PROGRAM MAIN
VAR
	test_bool:BOOL;
	test_int:INT;
	test_real:REAL;
	test_string:STRING;
	test_arr_int:ARRAY[1..10] OF INT;
	test_word:WORD;
	test_arr_bool:ARRAY[1..3] OF BOOL;
	test_structure:user_defined_structure;
	test_arr_string:ARRAY[1..3] OF STRING;
	
	fb_Time : FB_LocalSystemTime;

	byte1 : BYTE;
	string1 :STRING;

	
END_VAR

fb_Time(bEnable := TRUE); 

M_mappingIO();
M_measuringLC();
M_rfid();
runEveryCycle();
M_ReM();

METHOD M_mappingIO 
VAR_INPUT
END_VAR
GVL.fb_remIOmapping[0](iReM:= 0);
GVL.fb_remIOmapping[1](iReM:= 1);
GVL.fb_remIOmapping[2](iReM:= 2);
GVL.fb_remIOmapping[3](iReM:= 3);
GVL.fb_remIOmapping[4](iReM:= 4);
GVL.fb_remIOmapping[5](iReM:= 5);
GVL.fb_remIOmapping[6](iReM:= 6);
GVL.fb_remIOmapping[7](iReM:= 7);
GVL.fb_remIOmapping[8](iReM:= 8);
GVL.fb_remIOmapping[9](iReM:= 9);
GVL.fb_remAxisMapping[0](iReM :=0,iLift:=0,sNetID:='192.168.11.159.7.2',nSlaveAddr:=1002);
GVL.fb_remAxisMapping[1](iReM :=0,iLift:=1,sNetID:='192.168.11.159.7.2',nSlaveAddr:=1003);
GVL.fb_remAxisMapping[2](iReM :=1,iLift:=0,sNetID:='192.168.11.159.7.2',nSlaveAddr:=1006);
GVL.fb_remAxisMapping[3](iReM :=1,iLift:=1,sNetID:='192.168.11.159.7.2',nSlaveAddr:=1007);

GVL.fbAxisCtrl_Lift[0](stAxisCtrl:=GVL.stAxisCtrl_Lift[0],IN_OUT:=GVL.rem[0].lift[0].st_mcAxis);
GVL.fbAxisCtrl_Lift[1](stAxisCtrl:=GVL.stAxisCtrl_Lift[1],IN_OUT:=GVL.rem[0].lift[1].st_mcAxis);
GVL.fbAxisCtrl_Lift[2](stAxisCtrl:=GVL.stAxisCtrl_Lift[2],IN_OUT:=GVL.rem[1].lift[0].st_mcAxis);
GVL.fbAxisCtrl_Lift[3](stAxisCtrl:=GVL.stAxisCtrl_Lift[3],IN_OUT:=GVL.rem[1].lift[1].st_mcAxis);


GVL.fb_rmIOmapping[0](iRm:= 0);
GVL.fb_rmIOmapping[0](iRm:= 1);
GVL.fb_rmIOmapping[0](iRm:= 2);
GVL.fb_rmIOmapping[0](iRm:= 3);
GVL.fb_rmIOmapping[0](iRm:= 4);
//GVL.fb_pmAxisMapping[0](iPM :=0,iBuffer:=0,sNetID:='192.168.11.159.7.2',nSlaveAddr:=2002);
//GVL.fb_pmAxisMapping[1](iPM :=0,iBuffer:=1,sNetID:='192.168.11.159.7.2',nSlaveAddr:=2003);
//GVL.fb_pmAxisMapping[2](iPM :=1,iBuffer:=0,sNetID:='192.168.11.159.7.2',nSlaveAddr:=2006);
//GVL.fb_pmAxisMapping[3](iPM :=1,iBuffer:=1,sNetID:='192.168.11.159.7.2',nSlaveAddr:=2007);
GVL.fbAxisCtrl_Buffer[0](stAxisCtrl:=GVL.stAxisCtrl_Buffer[0],IN_OUT:=GVL.pm[0].buffer[0].st_mcAxis);
GVL.fbAxisCtrl_Buffer[1](stAxisCtrl:=GVL.stAxisCtrl_Buffer[1],IN_OUT:=GVL.pm[0].buffer[1].st_mcAxis);
GVL.fbAxisCtrl_Buffer[2](stAxisCtrl:=GVL.stAxisCtrl_Buffer[2],IN_OUT:=GVL.pm[1].buffer[0].st_mcAxis);
GVL.fbAxisCtrl_Buffer[3](stAxisCtrl:=GVL.stAxisCtrl_Buffer[3],IN_OUT:=GVL.pm[1].buffer[1].st_mcAxis);

(*GVL.arrSenDetect[1] := G_IO.arDI[4].Ch[0];
GVL.arrSenDetect[2] := G_IO.arDI[4].Ch[1];
GVL.arrSenDetect[3] := G_IO.arDI[4].Ch[2];
GVL.arrSenDetect[4] := G_IO.arDI[4].Ch[3];
GVL.arrSenDetect[5] := G_IO.arDI[4].Ch[4];*)

(*GVL.rem[0].infeed[0].roller.err						:= G_IO.arDI[0].Ch[0];
GVL.rem[0].infeed[0].valve_stopper.extended  		:= G_IO.arDI[0].Ch[1];
GVL.rem[0].infeed[0].valve_stopper.retracted  		:= G_IO.arDI[0].Ch[2];
GVL.rem[0].infeed[0].photo_sensor[0].set_status(G_IO.arDI[0].Ch[3],10,50);
GVL.rem[0].infeed[0].photo_sensor[1].set_status(G_IO.arDI[0].Ch[4],10,50);
GVL.rem[0].outfeed[0].roller.err					:= G_IO.arDI[0].Ch[5];
GVL.rem[0].outfeed[0].photo_sensor[0].set_status(G_IO.arDI[0].Ch[6],10,50);
GVL.rem[0].outfeed[0].photo_sensor[1].set_status(G_IO.arDI[0].Ch[7],10,50);
GVL.rem[0].lift[0].roller.err						:= G_IO.arDI[0].Ch[8];
GVL.rem[0].lift[0].contactor_axis						:= G_IO.arDI[0].Ch[9];
//GVL.rem[0].lift[0].limit_sensor[0]	:= TRUE;
//GVL.rem[0].lift[0].limit_sensor[1]	:= TRUE;
//GVL.rem[0].lift[0].limit_sensor[2]	:= TRUE;
GVL.rem[0].lift[0].limit_sensor[0]	:= G_IO.arDI[0].Ch[10];
GVL.rem[0].lift[0].limit_sensor[1]	:= G_IO.arDI[0].Ch[11];
GVL.rem[0].lift[0].limit_sensor[2]	:= G_IO.arDI[0].Ch[12];
GVL.rem[0].lift[0].valve_perturbation[0].extended  	:= G_IO.arDI[0].Ch[13];
GVL.rem[0].lift[0].valve_perturbation[0].retracted 	:= G_IO.arDI[0].Ch[14];
GVL.rem[0].lift[0].valve_perturbation[1].extended  	:= G_IO.arDI[0].Ch[15];
GVL.rem[0].lift[0].valve_perturbation[1].retracted 	:= G_IO.arDI[1].Ch[0];
GVL.rem[0].lift[0].valve_perturbation[2].extended  	:= G_IO.arDI[1].Ch[1];
GVL.rem[0].lift[0].valve_perturbation[2].retracted 	:= G_IO.arDI[1].Ch[2];
GVL.rem[0].lift[0].valve_perturbation[3].extended  	:= G_IO.arDI[1].Ch[3];
GVL.rem[0].lift[0].valve_perturbation[3].retracted	:= G_IO.arDI[1].Ch[4];
GVL.rem[0].lift[0].valve_clamp.extended  := G_IO.arDI[1].Ch[5];
GVL.rem[0].lift[0].valve_clamp.retracted  := G_IO.arDI[1].Ch[6];
GVL.rem[0].lift[0].photo_sensor[0].set_status(G_IO.arDI[1].Ch[7],10,50);
GVL.rem[0].lift[0].photo_sensor[1].set_status(G_IO.arDI[1].Ch[8],10,50);

G_IO.arDO[0].Ch[0]	:= GVL.rem[0].infeed[0].roller.Power;
G_IO.arDO[0].Ch[1]	:= GVL.rem[0].infeed[0].roller.forward;
G_IO.arDO[0].Ch[2]	:= GVL.rem[0].infeed[0].roller.backward;
G_IO.arDO[0].Ch[3]	:= GVL.rem[0].outfeed[0].roller.Power;
G_IO.arDO[0].Ch[4]	:= GVL.rem[0].outfeed[0].roller.forward;
G_IO.arDO[0].Ch[5]	:= GVL.rem[0].outfeed[0].roller.backward;
G_IO.arDO[0].Ch[6]	:= GVL.rem[0].lift[0].roller.Power;
G_IO.arDO[0].Ch[7]	:= GVL.rem[0].lift[0].roller.forward;
G_IO.arDO[0].Ch[8]	:= GVL.rem[0].lift[0].roller.backward;
G_IO.arDO[0].Ch[9]	:= GVL.rem[0].lift[0].power_axis;
G_IO.arDO[2].Ch[0]	:= GVL.rem[0].infeed[0].valve_stopper.extend;
G_IO.arDO[2].Ch[1]	:= GVL.rem[0].infeed[0].valve_stopper.retract;
G_IO.arDO[2].Ch[2]	:= GVL.rem[0].lift[0].valve_perturbation[0].extend;
G_IO.arDO[2].Ch[4]	:= GVL.rem[0].lift[0].valve_perturbation[1].extend;
G_IO.arDO[2].Ch[6]	:= GVL.rem[0].lift[0].valve_perturbation[2].extend;
G_IO.arDO[2].Ch[8]	:= GVL.rem[0].lift[0].valve_perturbation[3].extend;
G_IO.arDO[2].Ch[10]	:= GVL.rem[0].lift[0].valve_clamp.extend;
G_IO.arDO[2].Ch[11]	:= GVL.rem[0].lift[0].valve_clamp.retract;



GVL.rem[0].infeed[1].roller.err	:= G_IO.arDI[2].Ch[0];
GVL.rem[0].infeed[1].valve_stopper.extended  := G_IO.arDI[2].Ch[1];
GVL.rem[0].infeed[1].valve_stopper.retracted  := G_IO.arDI[2].Ch[2];
GVL.rem[0].infeed[1].photo_sensor[0].set_status(G_IO.arDI[2].Ch[3],10,50);
GVL.rem[0].infeed[1].photo_sensor[1].set_status(G_IO.arDI[2].Ch[4],10,50);
GVL.rem[0].outfeed[1].roller.err	:= G_IO.arDI[2].Ch[5];
GVL.rem[0].outfeed[1].photo_sensor[0].set_status(G_IO.arDI[2].Ch[6],10,50);
GVL.rem[0].outfeed[1].photo_sensor[1].set_status(G_IO.arDI[2].Ch[7],10,50);
GVL.rem[0].lift[1].roller.err	:= G_IO.arDI[2].Ch[8];
GVL.rem[0].lift[1].contactor_axis	:= G_IO.arDI[2].Ch[9];
//GVL.rem[0].lift[1].limit_sensor[0]	:= TRUE;
//GVL.rem[0].lift[1].limit_sensor[1]	:= TRUE;
//GVL.rem[0].lift[1].limit_sensor[2]	:= TRUE;
GVL.rem[0].lift[1].limit_sensor[0]	:= G_IO.arDI[2].Ch[10];
GVL.rem[0].lift[1].limit_sensor[1]	:= G_IO.arDI[2].Ch[11];
GVL.rem[0].lift[1].limit_sensor[2]	:= G_IO.arDI[2].Ch[12];
GVL.rem[0].lift[1].valve_perturbation[0].extended  := G_IO.arDI[2].Ch[13];
GVL.rem[0].lift[1].valve_perturbation[0].retracted  := G_IO.arDI[2].Ch[14];
GVL.rem[0].lift[1].valve_perturbation[1].extended  := G_IO.arDI[2].Ch[15];
GVL.rem[0].lift[1].valve_perturbation[1].retracted  := G_IO.arDI[3].Ch[0];
GVL.rem[0].lift[1].valve_perturbation[2].extended  := G_IO.arDI[3].Ch[1];
GVL.rem[0].lift[1].valve_perturbation[2].retracted  := G_IO.arDI[3].Ch[2];
GVL.rem[0].lift[1].valve_perturbation[3].extended  := G_IO.arDI[3].Ch[3];
GVL.rem[0].lift[1].valve_perturbation[3].retracted  := G_IO.arDI[3].Ch[4];
GVL.rem[0].lift[1].valve_clamp.extended  := G_IO.arDI[3].Ch[5];
GVL.rem[0].lift[1].valve_clamp.retracted  := G_IO.arDI[3].Ch[6];
GVL.rem[0].lift[1].photo_sensor[0].set_status(G_IO.arDI[3].Ch[7],10,50);
GVL.rem[0].lift[1].photo_sensor[1].set_status(G_IO.arDI[3].Ch[8],10,50);

G_IO.arDO[1].Ch[0]	:= GVL.rem[0].infeed[1].roller.Power;
G_IO.arDO[1].Ch[1]	:= GVL.rem[0].infeed[1].roller.forward;
G_IO.arDO[1].Ch[2]	:= GVL.rem[0].infeed[1].roller.backward;
G_IO.arDO[1].Ch[3]	:= GVL.rem[0].outfeed[1].roller.Power;
G_IO.arDO[1].Ch[4]	:= GVL.rem[0].outfeed[1].roller.forward;
G_IO.arDO[1].Ch[5]	:= GVL.rem[0].outfeed[1].roller.backward;
G_IO.arDO[1].Ch[6]	:= GVL.rem[0].lift[1].roller.Power;
G_IO.arDO[1].Ch[7]	:= GVL.rem[0].lift[1].roller.forward;
G_IO.arDO[1].Ch[8]	:= GVL.rem[0].lift[1].roller.backward;
G_IO.arDO[1].Ch[9]	:= GVL.rem[0].lift[1].power_axis;
G_IO.arDO[2].Ch[12]	:= GVL.rem[0].infeed[1].valve_stopper.extend;
G_IO.arDO[2].Ch[13]	:= GVL.rem[0].infeed[1].valve_stopper.retract;
G_IO.arDO[2].Ch[14]	:= GVL.rem[0].lift[1].valve_perturbation[0].extend;
G_IO.arDO[3].Ch[0]	:= GVL.rem[0].lift[1].valve_perturbation[1].extend;
G_IO.arDO[3].Ch[2]	:= GVL.rem[0].lift[1].valve_perturbation[2].extend;
G_IO.arDO[3].Ch[4]	:= GVL.rem[0].lift[1].valve_perturbation[3].extend;
G_IO.arDO[3].Ch[6]	:= GVL.rem[0].lift[1].valve_clamp.extend;
G_IO.arDO[3].Ch[7]	:= GVL.rem[0].lift[1].valve_clamp.retract;*)


//////////////////////////////PM[0]///////////////////////////////////
(*GVL.pm[0].buffer[0].contractor_axis				:= G_IO.arDI[50].Ch[0];
GVL.pm[0].buffer[0].axis_sensor					:= G_IO.arDI[50].Ch[1];
GVL.pm[0].buffer[0].surfae_slot_0				:= G_IO.arDI[50].Ch[2];
GVL.pm[0].buffer[0].surfae_slot_1				:= G_IO.arDI[50].Ch[3];
GVL.pm[0].buffer[0].surfae_slot_2				:= G_IO.arDI[50].Ch[4];
GVL.pm[0].buffer[0].above_fixture_light_curtain	:= G_IO.arDI[50].Ch[5];
GVL.pm[0].buffer[0].button						:= G_IO.arDI[50].Ch[6];
GVL.pm[0].buffer[0].locked						:= G_IO.arDI[50].Ch[7];
GVL.pm[0].buffer[0].magnet_locked				:= G_IO.arDI[50].Ch[8];
GVL.pm[0].buffer[1].contractor_axis				:= G_IO.arDI[50].Ch[9];
GVL.pm[0].buffer[1].axis_sensor					:= G_IO.arDI[50].Ch[10];
GVL.pm[0].buffer[1].surfae_slot_0				:= G_IO.arDI[50].Ch[11];
GVL.pm[0].buffer[1].surfae_slot_1				:= G_IO.arDI[50].Ch[12];
GVL.pm[0].buffer[1].surfae_slot_2				:= G_IO.arDI[50].Ch[13];
GVL.pm[0].buffer[1].above_fixture_light_curtain	:= G_IO.arDI[50].Ch[14];
GVL.pm[0].buffer[1].button						:= G_IO.arDI[50].Ch[15];
GVL.pm[0].buffer[1].locked						:= G_IO.arDI[51].Ch[0];
GVL.pm[0].buffer[1].magnet_locked				:= G_IO.arDI[51].Ch[1];
GVL.pm[0].contactor_robot						:= G_IO.arDI[51].Ch[2];
GVL.pm[0].inConv.valve[0].extended				:= G_IO.arDI[51].Ch[3];
GVL.pm[0].inConv.valve[0].retracted				:= G_IO.arDI[51].Ch[4];
GVL.pm[0].inConv.valve[1].extended				:= G_IO.arDI[51].Ch[5];
GVL.pm[0].inConv.valve[1].retracted				:= G_IO.arDI[51].Ch[6];
GVL.pm[0].inConv.valve[2].extended				:= G_IO.arDI[51].Ch[7];
GVL.pm[0].inConv.valve[2].retracted				:= G_IO.arDI[51].Ch[8];
GVL.pm[0].outConv.photo_sensor[0]				:= G_IO.arDI[51].Ch[9];
GVL.pm[0].outConv.photo_sensor[1]				:= G_IO.arDI[51].Ch[10];
GVL.pm[0].outConv.valve[0].extended				:= G_IO.arDI[51].Ch[11];
GVL.pm[0].outConv.valve[0].retracted			:= G_IO.arDI[51].Ch[12];
GVL.pm[0].outConv.valve[1].extended				:= G_IO.arDI[51].Ch[13];
GVL.pm[0].outConv.valve[1].retracted			:= G_IO.arDI[51].Ch[14];


GVL.pm[0].contactor_inConv						:= G_IO.arDI[54].Ch[0];//share with pm[1]
GVL.pm[0].contactor_inConv						:= G_IO.arDI[54].Ch[1];//share with pm[1]

G_IO.arDO[50].Ch[0]	:= GVL.pm[0].buffer[0].power_axis;
G_IO.arDO[50].Ch[1]	:= GVL.pm[0].buffer[0].magnet;
G_IO.arDO[50].Ch[2]	:= GVL.pm[0].buffer[1].power_axis;
G_IO.arDO[50].Ch[3]	:= GVL.pm[0].buffer[1].magnet;
G_IO.arDO[50].Ch[4]	:= GVL.pm[0].power_robot;
G_IO.arDO[50].Ch[12]	:= GVL.pm[0].buffer[0].lamp_button;
G_IO.arDO[50].Ch[13]	:= GVL.pm[0].buffer[1].lamp_button;

G_IO.arDO[52].Ch[0]	:= GVL.pm[0].inConv.valve[0].extend;
G_IO.arDO[52].Ch[2]	:= GVL.pm[0].inConv.valve[1].extend;
G_IO.arDO[52].Ch[4]	:= GVL.pm[0].inConv.valve[2].extend;
G_IO.arDO[52].Ch[6]	:= GVL.pm[0].outConv.valve[0].extend;
G_IO.arDO[52].Ch[8]	:= GVL.pm[0].outConv.valve[1].extend;

G_IO.arDO[50].Ch[10]	:= GVL.pm[0].power_inConv;//share with pm[1]
G_IO.arDO[50].Ch[11]	:= GVL.pm[0].power_outConv;//share with pm[1]
*)
END_METHOD

METHOD M_measuringLC : BOOL
VAR_INPUT
END_VAR

VAR
	i: INT;
	j: INT;
END_VAR
FOR i :=1 TO 32 DO
	GVL.ibyteNum[i] := i;
END_FOR
FOR i:=1 TO 32 DO	
	GVL.stMeasuringLC.arByte[i].Ch[0]	:= GVL.byteLC[i].0;
	GVL.stMeasuringLC.arByte[i].Ch[1]	:= GVL.byteLC[i].1;
	GVL.stMeasuringLC.arByte[i].Ch[2]	:= GVL.byteLC[i].2;
	GVL.stMeasuringLC.arByte[i].Ch[3]	:= GVL.byteLC[i].3;
	GVL.stMeasuringLC.arByte[i].Ch[4]	:= GVL.byteLC[i].4;
	GVL.stMeasuringLC.arByte[i].Ch[5]	:= GVL.byteLC[i].5;
	GVL.stMeasuringLC.arByte[i].Ch[6]	:= GVL.byteLC[i].6;
	GVL.stMeasuringLC.arByte[i].Ch[7]	:= GVL.byteLC[i].7;
END_FOR


GVL.stByte REF= GVL.stMeasuringLC;
END_METHOD

METHOD M_ReM : BOOL
VAR_INPUT
END_VAR

//========== Lift0 Axis Config ==========
(*GVL.rem[0].lift[0].mcAxis
(
	ZSN		:= GVL.rem[0].lift[0].limit_sensor[2] OR GVL.rem[0].lift[0].st_mcAxis.xHoming,
	ZSP		:= GVL.rem[0].lift[0].limit_sensor[1]	OR GVL.rem[0].lift[0].st_mcAxis.xHoming,
	IN_OUT	:= GVL.rem[0].lift[0].st_mcAxis, 
	AXIS	:= GVL.rem[0].lift[0].Axisref, 
);
GVL.rem[0].lift[0].st_mcAxis.bPosSensorShow	:= TRUE;
GVL.rem[0].lift[0].st_mcAxis.bNegSensorShow	:= TRUE;
GVL.rem[0].lift[0].st_mcAxis.bStopButtonShow	:= TRUE;
GVL.rem[0].lift[0].st_mcAxis.rMaxAcceleration	:= 50000;
GVL.rem[0].lift[0].st_mcAxis.rMaxDeceleration	:= 50000;
GVL.rem[0].lift[0].st_mcAxis.rMaxJerk			:= 500000;
GVL.rem[0].lift[0].st_mcAxis.rAcceleration	:= 2500;
GVL.rem[0].lift[0].st_mcAxis.rDeceleration	:= 2500;
GVL.rem[0].lift[0].st_mcAxis.rJerk			:= 12500;
GVL.rem[0].lift[0].st_mcAxis.rMaxVelocity		:= 100;
GVL.rem[0].lift[0].st_mcAxis.rMaxDistance		:= 50;
GVL.rem[0].lift[0].st_mcAxis.bPosSen	:= GVL.rem[0].lift[0].limit_sensor[1] ;
GVL.rem[0].lift[0].st_mcAxis.bNegSen	:= GVL.rem[0].lift[0].limit_sensor[2] ;
GVL.rem[0].lift[0].st_mcAxis.mcHome.bCalibrationCam	:= GVL.rem[0].lift[0].limit_sensor[0];
GVL.rem[0].lift[0].st_mcAxis.bPositionSensor	:= GVL.rem[0].lift[0].limit_sensor[0];
GVL.rem[0].lift[0].st_mcAxis.bdirFW	:= TRUE;
GVL.rem[0].lift[0].st_mcAxis.rSetPos	:= 0;
GVL.rem[0].lift[0].st_mcAxis.sNetID := '192.168.11.159.1.1';
GVL.rem[0].lift[0].st_mcAxis.nSlaveAddr	:= 1002;
//GVL.rem[0].lift[0].st_mcAxis.nSubIndex := 16#1F;
//GVL.rem[0].lift[0].st_mcAxis.nIndex	:= 16#2005;


//========== Lift1 Axis Config ==========
GVL.rem[0].lift[1].mcAxis
(
	ZSN		:= GVL.rem[0].lift[1].limit_sensor[2] OR GVL.rem[0].lift[1].st_mcAxis.xHoming,
	ZSP		:= GVL.rem[0].lift[1].limit_sensor[1]	OR GVL.rem[0].lift[1].st_mcAxis.xHoming,
	IN_OUT	:= GVL.rem[0].lift[1].st_mcAxis, 
	AXIS	:= GVL.rem[0].lift[1].Axisref, 
);
GVL.rem[0].lift[1].st_mcAxis.bPosSensorShow	:= TRUE;
GVL.rem[0].lift[1].st_mcAxis.bNegSensorShow	:= TRUE;
GVL.rem[0].lift[1].st_mcAxis.bStopButtonShow	:= TRUE;
GVL.rem[0].lift[1].st_mcAxis.rMaxAcceleration	:= 50000;
GVL.rem[0].lift[1].st_mcAxis.rMaxDeceleration	:= 50000;
GVL.rem[0].lift[1].st_mcAxis.rMaxJerk			:= 500000;
GVL.rem[0].lift[1].st_mcAxis.rAcceleration	:= 2500;
GVL.rem[0].lift[1].st_mcAxis.rDeceleration	:= 2500;
GVL.rem[0].lift[1].st_mcAxis.rJerk			:= 12500;
GVL.rem[0].lift[1].st_mcAxis.rMaxVelocity		:= 100;
GVL.rem[0].lift[1].st_mcAxis.rMaxDistance		:= 50;
GVL.rem[0].lift[1].st_mcAxis.bPosSen	:= GVL.rem[0].lift[1].limit_sensor[1] ;
GVL.rem[0].lift[1].st_mcAxis.bNegSen	:= GVL.rem[0].lift[1].limit_sensor[2] ;
GVL.rem[0].lift[1].st_mcAxis.mcHome.bCalibrationCam	:= GVL.rem[0].lift[1].limit_sensor[0];
GVL.rem[0].lift[1].st_mcAxis.bPositionSensor	:= GVL.rem[0].lift[1].limit_sensor[0];
GVL.rem[0].lift[1].st_mcAxis.bdirFW	:= TRUE;
GVL.rem[0].lift[1].st_mcAxis.rSetPos	:= 0;
GVL.rem[0].lift[1].st_mcAxis.sNetID := '192.168.11.159.1.1';
GVL.rem[0].lift[1].st_mcAxis.nSlaveAddr	:= 1003;
//GVL.rem[0].lift[1].st_mcAxis.nSubIndex := 16#1F;
//GVL.rem[0].lift[1].st_mcAxis.nIndex	:=  16#2005;

CASE GVL.iFRtest OF 
	0:		
		//IF GVL.rem[0].lift[0].st_mcAxis.xHomingDone THEN
			IF GVL.bTs1 THEN
				GVL.rem[0].lift[0].st_mcAxis.mcMoveAbsolute.Execute := FALSE;
				GVL.iFRtest :=1;
			END_IF
		//END_IF
	1://open positon
		GVL.rem[0].lift[0].st_mcAxis.rActualPosSet := 0;
		GVL.rem[0].lift[0].st_mcAxis.rVelocitySet := 300;			
		GVL.rem[0].lift[0].st_mcAxis.mcMoveAbsolute.Execute := TRUE;
		GVL.rem[0].lift[1].st_mcAxis.rActualPosSet := 0;
		GVL.rem[0].lift[1].st_mcAxis.rVelocitySet := 300;			
		GVL.rem[0].lift[1].st_mcAxis.mcMoveAbsolute.Execute := TRUE;
		IF GVL.rem[0].lift[0].st_mcAxis.mcMoveAbsolute.Done AND GVL.rem[0].lift[1].st_mcAxis.mcMoveAbsolute.Done THEN
			GVL.rem[0].lift[0].st_mcAxis.mcMoveAbsolute.Execute := FALSE;
			GVL.rem[0].lift[1].st_mcAxis.mcMoveAbsolute.Execute := FALSE;
			GVL.iFRtest := 2;
		END_IF
	
	2:
		ton_delay.IN := TRUE;
		IF ton_delay.Q THEN
			ton_delay.IN := FALSE;
			GVL.iFRtest := 3;
		END_IF
	3://close position
		GVL.rem[0].lift[0].st_mcAxis.rActualPosSet := 424;
		GVL.rem[0].lift[0].st_mcAxis.rVelocitySet := 300;			
		GVL.rem[0].lift[0].st_mcAxis.mcMoveAbsolute.Execute := TRUE;
		GVL.rem[0].lift[1].st_mcAxis.rActualPosSet := 424;
		GVL.rem[0].lift[1].st_mcAxis.rVelocitySet := 300;			
		GVL.rem[0].lift[1].st_mcAxis.mcMoveAbsolute.Execute := TRUE;		
		GVL.st_mcAxis[1].mcMoveAbsolute.Execute := TRUE;
			IF GVL.rem[0].lift[0].st_mcAxis.mcMoveAbsolute.Done AND GVL.rem[0].lift[1].st_mcAxis.mcMoveAbsolute.Done THEN
				GVL.rem[0].lift[0].st_mcAxis.mcMoveAbsolute.Execute := FALSE;
				GVL.rem[0].lift[1].st_mcAxis.mcMoveAbsolute.Execute := FALSE;
				GVL.iFRtest := 4;
			END_IF   
	4://delay
		ton_delay.IN := TRUE;
		IF ton_delay.Q THEN
			ton_delay.IN := FALSE;
			GVL.iFRtest := 5;
		END_IF
	5://open positon
		GVL.rem[0].lift[0].st_mcAxis.rActualPosSet := 0;
		GVL.rem[0].lift[0].st_mcAxis.rVelocitySet := 300;			
		GVL.rem[0].lift[0].st_mcAxis.mcMoveAbsolute.Execute := TRUE;
		GVL.rem[0].lift[1].st_mcAxis.rActualPosSet := 0;
		GVL.rem[0].lift[1].st_mcAxis.rVelocitySet := 300;			
		GVL.rem[0].lift[1].st_mcAxis.mcMoveAbsolute.Execute := TRUE;
		IF GVL.rem[0].lift[0].st_mcAxis.mcMoveAbsolute.Done AND GVL.rem[0].lift[1].st_mcAxis.mcMoveAbsolute.Done THEN
			GVL.rem[0].lift[0].st_mcAxis.mcMoveAbsolute.Execute := FALSE;
			GVL.rem[0].lift[1].st_mcAxis.mcMoveAbsolute.Execute := FALSE;
			GVL.iFRtest := 6;
		END_IF
	6:
		GVL.iFRtest := 0;
END_CASE*)
END_METHOD

METHOD M_rfid : BOOL
VAR_INPUT
END_VAR

VAR
	i: INT;
	
END_VAR
byte1 := ASC(string1);
FOR i:=0 TO 3 DO	
	GVL.arIn[i].Ch[0]	:= GVL.rfidIn[i].0;
	GVL.arIn[i].Ch[1]	:= GVL.rfidIn[i].1;
	GVL.arIn[i].Ch[2]	:= GVL.rfidIn[i].2;
	GVL.arIn[i].Ch[3]	:= GVL.rfidIn[i].3;
	GVL.arIn[i].Ch[4]	:= GVL.rfidIn[i].4;
	GVL.arIn[i].Ch[5]	:= GVL.rfidIn[i].5;
	GVL.arIn[i].Ch[6]	:= GVL.rfidIn[i].6;
	GVL.arIn[i].Ch[7]	:= GVL.rfidIn[i].7;
	GVL.rfidOut[i].0	:= GVL.arOut[i].Ch[0];
	GVL.rfidOut[i].1	:= GVL.arOut[i].Ch[1];
	GVL.rfidOut[i].2	:= GVL.arOut[i].Ch[2];
	GVL.rfidOut[i].3	:= GVL.arOut[i].Ch[3];
	GVL.rfidOut[i].4	:= GVL.arOut[i].Ch[4];
	GVL.rfidOut[i].5	:= GVL.arOut[i].Ch[5];
	GVL.rfidOut[i].6	:= GVL.arOut[i].Ch[6];
	GVL.rfidOut[i].7	:= GVL.arOut[i].Ch[7];	
END_FOR

FOR i:=4 TO 31 DO
	GVL.rfidOut[i] := INT_TO_BYTE(28*GVL.n+i-3);
END_FOR
END_METHOD

METHOD runEveryCycle : BOOL
VAR_INPUT
END_VAR

VAR
	


END_VAR
(*
CASE GVL.iFRtest OF 
	0:		
		IF GVL.st_mcAxis[0].xHomingDone THEN
			IF GVL.bTs1 THEN
				GVL.st_mcAxis[0].mcMoveAbsolute.Execute := FALSE;
				GVL.iFRtest :=1;
			END_IF
		END_IF
		IF GVL.bBeltTs THEN
			G_IO.arDI[5].Ch[2] := TRUE;
			G_IO.arDI[5].Ch[3] := TRUE;
			GVL.st_mcAxis[0].mcMoveAbsolute.Execute := FALSE;
			GVL.iFRtest :=100;
		END_IF
	100:
		GVL.st_mcAxis[0].rActualPosSet := 60000000;
		GVL.st_mcAxis[0].rVelocitySet := 150;	
		GVL.st_mcAxis[0].mcMoveAbsolute.Execute := TRUE;	
		IF NOT GVL.bBeltTs THEN
			GVL.st_mcAxis[0].mcMoveAbsolute.Execute := FALSE;
			GVL.st_mcAxis[0].mcStop.Execute := TRUE;
			IF GVL.st_mcAxis[0].mcStop.Done THEN
				GVL.st_mcAxis[0].mcStop.Execute := FALSE;
				GVL.iFRtest :=0;
			END_IF
			
		END_IF
	1://open positon
		valve := FALSE;
		IF retracted THEN
			GVL.st_mcAxis[0].rActualPosSet := 102.8;
			GVL.st_mcAxis[0].rVelocitySet := 300;			
			GVL.st_mcAxis[0].mcMoveAbsolute.Execute := TRUE;
			IF GVL.st_mcAxis[0].mcMoveAbsolute.Done THEN
				GVL.st_mcAxis[0].mcMoveAbsolute.Execute := FALSE;
				GVL.iFRtest := 2;
			END_IF
		END_IF
	2://valve extend
		valve := TRUE;
		IF extended THEN
			GVL.iFRtest := 3;
		END_IF
	3://delay
		ton_delay.IN := TRUE;
		IF ton_delay.Q THEN
			ton_delay.IN := FALSE;
			GVL.iFRtest := 4;
		END_IF
	4://close position
		GVL.st_mcAxis[0].rActualPosSet := -78.4;
		GVL.st_mcAxis[0].rVelocitySet := 300;			
		GVL.st_mcAxis[0].mcMoveAbsolute.Execute := TRUE;
		IF GVL.st_mcAxis[0].mcMoveAbsolute.Done THEN
			GVL.st_mcAxis[0].mcMoveAbsolute.Execute := FALSE;
			GVL.iFRtest := 6;
		END_IF	   
	5://delay
		ton_delay.IN := TRUE;
		IF ton_delay.Q THEN
			ton_delay.IN := FALSE;
			GVL.iFRtest := 6;
		END_IF
	6://valve retract
		valve := FALSE;
		IF retracted THEN
			GVL.iFRtest := 7;
		END_IF	
	7://valve extend
		valve := TRUE;
		IF extended THEN
			GVL.iFRtest := 8;
		END_IF	
	8://delay
		ton_delay.IN := TRUE;
		IF ton_delay.Q THEN
			ton_delay.IN := FALSE;
			GVL.iFRtest := 9;
		END_IF
	9://open positon
		GVL.st_mcAxis[0].rActualPosSet := 102.8;
		GVL.st_mcAxis[0].rVelocitySet := 300;			
		GVL.st_mcAxis[0].mcMoveAbsolute.Execute := TRUE;
		IF GVL.st_mcAxis[0].mcMoveAbsolute.Done THEN
			GVL.st_mcAxis[0].mcMoveAbsolute.Execute := FALSE;
			GVL.iFRtest := 10;
		END_IF
	10:
		GVL.iFRtest := 0;
END_CASE
*)
END_METHOD

END_PROGRAM

(* stored: Version 1.1.0.1, ProductVersion 3.1.4024.12
   POU MAIN: Id {79b373eb-1c8e-4458-8b04-107fcef16361}, SpecialFunc None
   Method M_mappingIO: Id {e0caa2a2-200b-484a-9495-8cf8901a2628}
   Method M_measuringLC: Id {d676c292-2f0e-482c-8f77-a1f869b0f883}
   Method M_ReM: Id {64ae7519-e3a0-402c-ae7d-63672adcb499}
   Method M_rfid: Id {5c57c28f-978a-4ef1-8020-2ee35fe2b4f0}
   Method runEveryCycle: Id {79ccd451-642e-4685-afbb-6dd16a84c35a} *)
